# EPICS autosave request: iocBoot/gmca_23i_ioc2/dbSave/robot.req
% $(P)pause
$(P)gh_pos
$(P)gy_pos
$(P)tmoh
$(P)senh
$(P)senb
$(P)senc
$(P)send
$(P)senb_extradelay
$(P)warmup_duration
